// TwinCAT 3 PLC project B1RollingAverage_Plc
// Title: B1RollingAverage_Plc
// Company: Tc3 Project
// ProjectVersion: 1.0.0.0
// ProgramVersion: 3.1.4026.22
// libraries:
//   Tc2_Standard, * (Beckhoff Automation GmbH)
//   Tc2_System, * (Beckhoff Automation GmbH)
// project tree:
//   / PlcTask.TcTTO
//   POUs/ FB_RollingAverage.TcPOU, MAIN.TcPOU
// real-time tasks:
//   TASK PlcTask: cycle T#10ms, priority 20, ADS port 350

CONFIGURATION B1RollingAverage_Plc
    RESOURCE PLC ON TwinCAT3
        TASK PlcTask(INTERVAL := T#10ms, PRIORITY := 20);
        PROGRAM MAIN WITH PlcTask : MAIN;
    END_RESOURCE
END_CONFIGURATION

// ---- POUs/MAIN.TcPOU
PROGRAM MAIN
VAR
END_VAR

END_PROGRAM

// ---- POUs/FB_RollingAverage.TcPOU
FUNCTION_BLOCK FB_RollingAverage
VAR
    samples : ARRAY[0..15] OF INT;
    sampleCount : INT := 8;
    nextIndex : INT;
END_VAR

METHOD Step : INT
VAR_INPUT
    sample : INT;
END_VAR
VAR
    sum : DINT;
    i : INT;
END_VAR
samples[nextIndex] := sample;
nextIndex := (nextIndex + 1) MOD sampleCount;
sum := 0;
FOR i := 1 TO sampleCount DO
    sum := sum + samples[i];
END_FOR
Step := DINT_TO_INT(sum / sampleCount);
END_METHOD

END_FUNCTION_BLOCK
